// TIA Portal V16 export
// export: Created 2023-11-14T19:43:16.1887639Z, ExportSetting WithDefaults, DisplayName Totally Integrated Automation Portal, DisplayVersion V16, DisplayName TIA Portal Version Control Interface, DisplayVersion V16, DisplayName TIA Portal Openness, DisplayVersion V16, DisplayName SINAMICS Startdrive Advanced, DisplayVersion V16, DisplayName SINAMICS Startdrive G130, G150, S120, S150, SINAMICS MV, S210, DisplayVersion V16, DisplayName SINAMICS Startdrive G110M, G120, G120C, G120D, G120P, DisplayVersion V16, DisplayName STEP 7 Professional, DisplayVersion V16, DisplayName STEP 7 Safety, DisplayVersion V16, DisplayName WinCC Professional, DisplayVersion V16
DATA_BLOCK "DATOS_MODSEC"   // DB13
{ S7_Optimized_Access := 'TRUE' }
VERSION : 0.1
// stored: AutoNumber true, DBAccessibleFromOPCUA true, IsOnlyStoredInLoadMemory false, IsRetainMemResEnabled false, IsWriteProtectedInAS false, MemoryReserve 100
   VAR
      SimuHR : Int;
   END_VAR
   VAR RETAIN
      "Paso Control HR" : Time := T#5000ms;
      "Paso Grafica" : Time := T#10ms;
      "CRECIMIENTO HR" : Real := 80.0;
      TempMinHR : Real := 22.0;
   END_VAR
   VAR
      TempInf : Real := 0.0;
      TempSup : Real := 100.0;
      TempFilt : Real;
      TempFiltJP : Real;
      HRAux : Real;
      HRAuxJP : Real;
      HRFilt : Real;
      HRSim : Int;
      TempSim : Int;
      ProporcionHumedad : Real := 0.9;
      TempFiltCuar : Real;
      HRFiltCuar : Real;
      HRAuxCuar : Real;
   END_VAR
BEGIN
END_DATA_BLOCK
